TYPE PositionExtremaStruct :
STRUCT
  minimum, maximum : LREAL;
  t_min, t_max : LREAL;  
END_STRUCT
END_TYPE

(* stored: Version 1.1.0.1, ProductVersion 3.1.4024.6
   DUT PositionExtremaStruct: Id {b615dcba-8544-436f-9a57-30985945064e} *)
